// Provides acces to control the light tower components.
FUNCTION_BLOCK FB_LightTower
VAR
	_redLight		: FB_LightTowerComponent;
	_yellowLight	: FB_LightTowerComponent;
	_greenLight		: FB_LightTowerComponent;
	RtrigBuzzer		: R_TRIG;
END_VAR

VAR_INPUT
	bBuzzerTrigger	: BOOL;
	bBuzzerReset	: BOOL;
END_VAR

VAR_OUTPUT
	bBuzzerOut	: BOOL;
END_VAR

RtrigBuzzer(
	CLK := bBuzzerTrigger);

IF RtrigBuzzer.Q THEN
	bBuzzerOut := TRUE;
END_IF

IF bBuzzerReset THEN
	bBuzzerOut := FALSE;
END_IF
	
_redLight();
_yellowLight();
_greenLight();

PROPERTY GreenLight : I_LightTowerComponent
GET
GreenLight := _greenLight;
END_GET
END_PROPERTY

PROPERTY OrangeLight : I_LightTowerComponent
GET
OrangeLight := _yellowLight;
END_GET
END_PROPERTY

PROPERTY RedLight : I_LightTowerComponent
GET
RedLight := _redLight;
END_GET
END_PROPERTY

END_FUNCTION_BLOCK

(* stored: Version 1.1.0.1, ProductVersion 3.1.4024.13
   POU FB_LightTower: Id {8b6b0bb1-2528-035e-0ba1-b7066ca640fc}, SpecialFunc None
   Property GreenLight: Id {e65e7007-9a97-048f-308c-acb6806aea44}
   Get Get: Id {e1673a8a-1b77-00de-2e8e-077f922bbbfa}
   Property OrangeLight: Id {ebf94a05-c1b3-0586-0156-2445e6a0c2cf}
   Get Get: Id {12cb6937-e688-057b-057b-f10dadbdd932}
   Property RedLight: Id {83ece07b-b76f-0f56-1233-170ee7e5864b}
   Get Get: Id {2880d581-3fc0-038f-20f2-9eb952a5f265} *)
